Staubli VAL3: DealRobMaster.dtx

mdesc mNomSpeed
public string sFileList
public string sDeli[4]
  [0] = "A"
  [1] = "C"
  [2] = "B"
  [3] = "D"
bool bUserRefresh
bool bListRefresh
bool bExit
num nSelected
string sItem
string sFolder = "Disk://robmaster/"
string sOutputFolder = "Disk://Traj/"
string sFileTemp
frame fFrame = {fatherId=world[0]}
tool tTool = {fatherId=flange[0], ioLink=valve1}
